// TIA Portal project "Clase2" (V14)
// Equivalente del tutorial 1 del TIA Portal de Youtube

(* hardware
DEVICE "S7-1200 station_1"  S7-1200 Station
   slot 0: "Rack_0"  S7-1200 Rack  Rack  V1.0
   slot 1: "Limon_PLC"  CPU 1214C DC/DC/DC  6ES7 214-1AG40-0XB0  V4.2
DEVICE "S71500/ET200MP station_1"  S7-1500 station
   slot 0: "Rail_0"  Rack  6ES7 590-1***0-0AA0
   slot 1: "Limon 1516"  CPU 1516F-3 PN/DP  6ES7 516-3FN01-0AB0  V2.1
      slot 3: "CPU display_1"  6ES7591-1BA00-0AA0
   slot 2: "DI 32x24VDC HF_1"  DI 32x24VDC HF  6ES7 521-1BL00-0AB0  V2.1
   slot 3: "DQ 32x24VDC/0.5A HF_1"  DQ 32x24VDC/0.5A HF  6ES7 522-1BL01-0AB0  V1.0
DEVICE "S71500/ET200MP station_2"  S7-1500 station
   slot 0: "Rail_0"  Rack  6ES7 590-1***0-0AA0
   slot 1: "PLC_1"  Unspecific CPU 1500  6ES7 5XX-XXXXX-XXXX  V2.1
*)

// ===== PLC "Limon_PLC"  CPU 1214C DC/DC/DC =====

VAR_GLOBAL   // PLC tag table "Default tag table"
   "start" AT %I0.0 : Bool;
   "stop" AT %I0.1 : Bool;
   "L1" AT %Q0.0 : Bool;
   "L2" AT %Q0.1 : Bool;
   "variable" AT %M2.0 : Bool;
END_VAR

// folder: System blocks/Program resources

DATA_BLOCK "Timer1"   // DB1
{ S7_Optimized_Access := 'TRUE' }
AUTHOR : Simatic
FAMILY : IEC
NAME : IEC_TMR
VERSION : 1.0
// stored: InstanceOfName IEC_TIMER
"IEC_TIMER"
BEGIN
END_DATA_BLOCK

DATA_BLOCK "Timer2"   // DB2
{ S7_Optimized_Access := 'TRUE' }
AUTHOR : Simatic
FAMILY : IEC
NAME : IEC_TMR
VERSION : 1.0
// stored: InstanceOfName IEC_TIMER
"IEC_TIMER"
BEGIN
END_DATA_BLOCK

// folder: (top level)

FUNCTION "Arranque_Paro" : Void   // FC1, LAD
TITLE = Arranque y Paro
{ S7_Optimized_Access := 'TRUE' }
VERSION : 0.1
// Demostración de encendido y apagado de una lámpara con enclavamiento.
BEGIN

REGION Network 1: L1
   // Lámpara 1
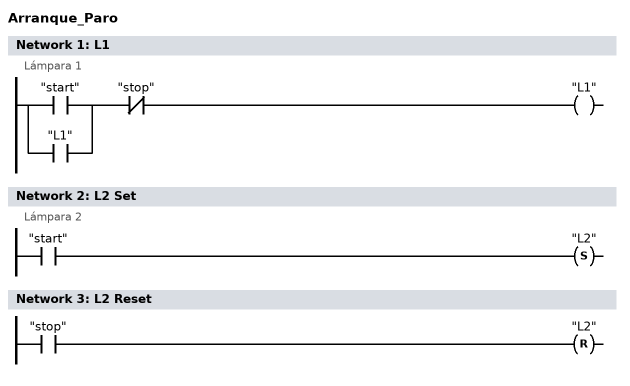
   RUNG wire#powerrail
      Contact( "start" )
      wire#w1
      I_Contact( "stop" )
      Coil( "L1" )
   END_RUNG
   RUNG wire#powerrail
      Contact( "L1" )
   END_RUNG wire#w1
   // the same network as SCL:
   "L1" := ("start" OR "L1") AND NOT "stop";
END_REGION

REGION Network 2: L2 Set
   // Lámpara 2
   RUNG wire#powerrail
      Contact( "start" )
      S_Coil( "L2" )
   END_RUNG
   // the same network as SCL:
   IF "start" THEN "L2" := TRUE; END_IF;
END_REGION

REGION Network 3: L2 Reset
   RUNG wire#powerrail
      Contact( "stop" )
      R_Coil( "L2" )
   END_RUNG
   // the same network as SCL:
   IF "stop" THEN "L2" := FALSE; END_IF;
END_REGION
END_FUNCTION

FUNCTION "Temporizadores" : Void   // FC2, LAD
{ S7_Optimized_Access := 'TRUE' }
VERSION : 0.1
BEGIN

REGION Network 1
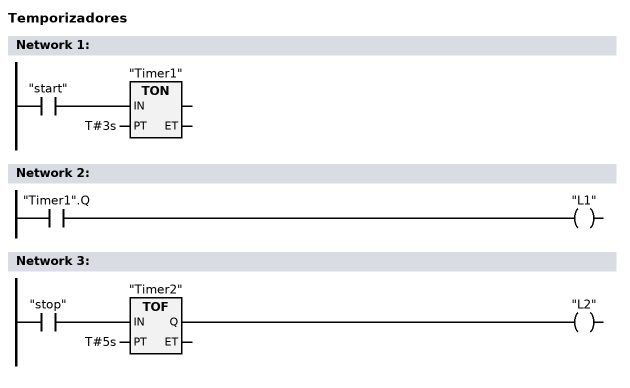
   "Timer1".TON(IN := "start", PT := T#3s);
END_REGION

REGION Network 2
   RUNG wire#powerrail
      Contact( "Timer1".Q )
      Coil( "L1" )
   END_RUNG
   // the same network as SCL:
   "L1" := "Timer1".Q;
END_REGION

REGION Network 3
   "Timer2".TOF(IN := "stop", PT := T#5s);
   "L2" := "Timer2".Q;
END_REGION
END_FUNCTION

ORGANIZATION_BLOCK "Main"   // OB1, LAD, ProgramCycle
TITLE = "Main Program Sweep (Cycle)"
{ S7_Optimized_Access := 'TRUE' }
VERSION : 0.1
   VAR_INPUT
      Initial_Call : Bool;   // Initial call of this OB
      Remanence : Bool;   // =True, if remanent data are available
   END_VAR
BEGIN

REGION Network 1
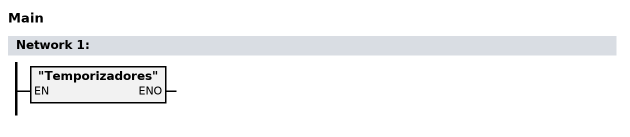
   RUNG wire#powerrail
      "Temporizadores"()
   END_RUNG
   // the same network as SCL:
   "Temporizadores"();
END_REGION
END_ORGANIZATION_BLOCK

// ===== PLC "Limon 1516"  CPU 1516F-3 PN/DP =====

VAR_GLOBAL   // PLC tag table "Default tag table"
   "start" AT %I0.0 : Bool;
   "stop" AT %I0.1 : Bool;
   "L1" AT %Q0.0 : Bool;
   "L2" AT %Q0.1 : Bool;
   "variable" AT %M2.0 : Bool;
END_VAR

// folder: System blocks/Program resources

DATA_BLOCK "Timer1"   // DB1
{ S7_Optimized_Access := 'TRUE' }
AUTHOR : Simatic
FAMILY : IEC
NAME : IEC_TMR
VERSION : 1.0
// stored: InstanceOfName IEC_TIMER
"IEC_TIMER"
BEGIN
END_DATA_BLOCK

DATA_BLOCK "Timer2"   // DB2
{ S7_Optimized_Access := 'TRUE' }
AUTHOR : Simatic
FAMILY : IEC
NAME : IEC_TMR
VERSION : 1.0
// stored: InstanceOfName IEC_TIMER
"IEC_TIMER"
BEGIN
END_DATA_BLOCK

// folder: (top level)

FUNCTION "Arranque_Paro" : Void   // FC1, LAD
TITLE = Arranque y Paro
{ S7_Optimized_Access := 'TRUE' }
VERSION : 0.1
// Demostración de encendido y apagado de una lámpara con enclavamiento.
BEGIN

REGION Network 1: L1
   // Lámpara 1
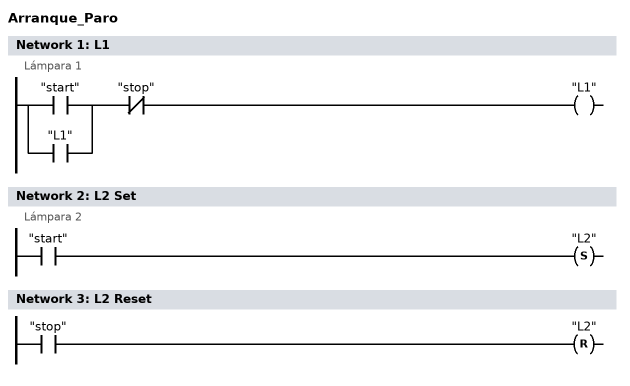
   RUNG wire#powerrail
      Contact( "start" )
      wire#w1
      I_Contact( "stop" )
      Coil( "L1" )
   END_RUNG
   RUNG wire#powerrail
      Contact( "L1" )
   END_RUNG wire#w1
   // the same network as SCL:
   "L1" := ("start" OR "L1") AND NOT "stop";
END_REGION

REGION Network 2: L2 Set
   // Lámpara 2
   RUNG wire#powerrail
      Contact( "start" )
      S_Coil( "L2" )
   END_RUNG
   // the same network as SCL:
   IF "start" THEN "L2" := TRUE; END_IF;
END_REGION

REGION Network 3: L2 Reset
   RUNG wire#powerrail
      Contact( "stop" )
      R_Coil( "L2" )
   END_RUNG
   // the same network as SCL:
   IF "stop" THEN "L2" := FALSE; END_IF;
END_REGION
END_FUNCTION

FUNCTION "Temporizadores" : Void   // FC2, LAD
TITLE = Uso de Temporizadores
{ S7_Optimized_Access := 'TRUE' }
VERSION : 0.1
BEGIN

REGION Network 1: TON
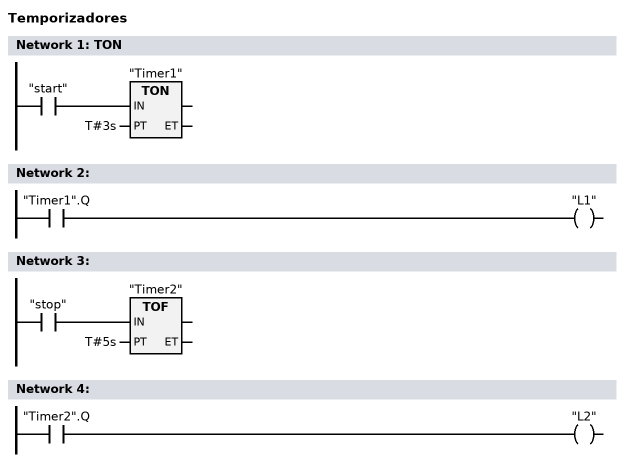
   "Timer1".TON(IN := "start", PT := T#3s);
END_REGION

REGION Network 2
   RUNG wire#powerrail
      Contact( "Timer1".Q )
      Coil( "L1" )
   END_RUNG
   // the same network as SCL:
   "L1" := "Timer1".Q;
END_REGION

REGION Network 3
   "Timer2".TOF(IN := "stop", PT := T#5s);
END_REGION

REGION Network 4
   RUNG wire#powerrail
      Contact( "Timer2".Q )
      Coil( "L2" )
   END_RUNG
   // the same network as SCL:
   "L2" := "Timer2".Q;
END_REGION
END_FUNCTION

ORGANIZATION_BLOCK "Main"   // OB1, LAD, ProgramCycle
TITLE = "Main Program Sweep (Cycle)"
{ S7_Optimized_Access := 'TRUE' }
VERSION : 0.1
   VAR_INPUT
      Initial_Call : Bool;   // Initial call of this OB
      Remanence : Bool;   // =True, if remanent data are available
   END_VAR
BEGIN

REGION Network 1
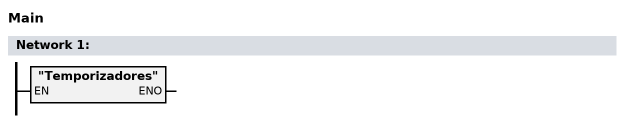
   RUNG wire#powerrail
      "Temporizadores"()
   END_RUNG
   // the same network as SCL:
   "Temporizadores"();
END_REGION
END_ORGANIZATION_BLOCK

// ===== PLC "PLC_1"  Unspecific CPU 1500 =====

ORGANIZATION_BLOCK "Main"   // OB1, LAD, ProgramCycle
TITLE = "Main Program Sweep (Cycle)"
{ S7_Optimized_Access := 'TRUE' }
VERSION : 0.1
   VAR_INPUT
      Initial_Call : Bool;   // Initial call of this OB
      Remanence : Bool;   // =True, if remanent data are available
   END_VAR
BEGIN
END_ORGANIZATION_BLOCK